FUNCTION_BLOCK F_GetItemAITests EXTENDS TcUnit.FB_TestSuite

VAR
	
	(* In/Out test*)		
	
END_VAR



//==============================================================
//01.CASE_Code
//==============================================================
Case_code01_GTIN_extractedWrong();
Case_code02_SERIAL_extractedWrong();
Case_code03_RSKU_extractedWrong();
Case_code04_BATCH_extractedWrong();
Case_code05_PO_extractedWrong();

//==============================================================
//02.Outer_Code
//==============================================================


//==============================================================
//03.Pack_Code
//==============================================================

METHOD INTERNAL Case_code01_GTIN_extractedWrong
VAR
	sFullCode		: T_MaxString;
	eCodeType		: CODE.E_CodeAI;
	stCodeInfo		: CODE.ST_CodeInfo;
	
	sF_GetItemAI	: T_MaxString;	
END_VAR
// Validation data init
stCodeInfo.eCodeType	:= CODE.E_CodeType.E_CASE;
TestInit(eCodeType := eCodeType, sFullCode := sFullcode, stCodeInfo := stCodeInfo);

//Change some data for test scenario below
sFullCode := '(01)17501031711052(21)86174He081137058500(240)10108245(10)86352024(91)5304012';
eCodeType	:= CODE.E_CodeAI.GTIN;


	
TcUnit.TEST('Case_code01_GTIN_extractedWrong');

	sF_GetItemAI := CODE.F_GetItemAI(sFullCode := sFullCode, 
									 eCodeType := eCodeType, 
									 stCodeInfo := stCodeInfo);
	
	AssertEquals_STRING(Expected:= '17501031711052', 
						Actual:= TO_STRING(sF_GetItemAI), 
						Message:= 'Wrong GTIN extracted');						

TEST_FINISHED();
END_METHOD

METHOD INTERNAL Case_code02_SERIAL_extractedWrong
VAR
	sFullCode		: T_MaxString;
	eCodeType		: CODE.E_CodeAI;
	stCodeInfo		: CODE.ST_CodeInfo;
	
	sF_GetItemAI	: T_MaxString;	
END_VAR
// Validation data init
stCodeInfo.eCodeType	:= CODE.E_CodeType.E_CASE;
TestInit(eCodeType := eCodeType, sFullCode := sFullcode, stCodeInfo := stCodeInfo);

//Change some data for test scenario below
sFullCode := '(01)17501031711052(21)86174He081137058500(240)10108245(10)86352024(91)5304012';
eCodeType	:= CODE.E_CodeAI.SERIAL;


	
TcUnit.TEST('Case_code02_SERIAL_extractedWrong');

	sF_GetItemAI := CODE.F_GetItemAI(sFullCode := sFullCode, 
									 eCodeType := eCodeType, 
									 stCodeInfo := stCodeInfo);
	
	AssertEquals_STRING(Expected:= '86174He081137058500', 
						Actual:= TO_STRING(sF_GetItemAI), 
						Message:= 'Wrong SERIAL extracted');						

TEST_FINISHED();
END_METHOD

METHOD INTERNAL Case_code03_RSKU_extractedWrong
VAR
	sFullCode		: T_MaxString;
	eCodeType		: CODE.E_CodeAI;
	stCodeInfo		: CODE.ST_CodeInfo;
	
	sF_GetItemAI	: T_MaxString;	
END_VAR
// Validation data init
stCodeInfo.eCodeType	:= CODE.E_CodeType.E_CASE;
TestInit(eCodeType := eCodeType, sFullCode := sFullcode, stCodeInfo := stCodeInfo);

//Change some data for test scenario below
sFullCode := '(01)17501031711052(21)86174He081137058500(240)10108245(10)86352024(91)5304012';
eCodeType	:= CODE.E_CodeAI.RSKU;


	
TcUnit.TEST('Case_code03_RSKU_extractedWrong');

	sF_GetItemAI := CODE.F_GetItemAI(sFullCode := sFullCode, 
									 eCodeType := eCodeType, 
									 stCodeInfo := stCodeInfo);
	
	AssertEquals_STRING(Expected:= '10108245', 
						Actual:= TO_STRING(sF_GetItemAI), 
						Message:= 'Wrong RSKU extracted');						

TEST_FINISHED();
END_METHOD

METHOD INTERNAL Case_code04_BATCH_extractedWrong
VAR
	sFullCode		: T_MaxString;
	eCodeType		: CODE.E_CodeAI;
	stCodeInfo		: CODE.ST_CodeInfo;
	
	sF_GetItemAI	: T_MaxString;	
END_VAR
// Validation data init
stCodeInfo.eCodeType	:= CODE.E_CodeType.E_CASE;
TestInit(eCodeType := eCodeType, sFullCode := sFullcode, stCodeInfo := stCodeInfo);

//Change some data for test scenario below
sFullCode := '(01)17501031711052(21)86174He081137058500(240)10108245(10)86352024(91)5304012';
eCodeType	:= CODE.E_CodeAI.BATCH;


	
TcUnit.TEST('Case_code04_BATCH_extractedWrong');

	sF_GetItemAI := CODE.F_GetItemAI(sFullCode := sFullCode, 
									 eCodeType := eCodeType, 
									 stCodeInfo := stCodeInfo);
	
	AssertEquals_STRING(Expected:= '86352024', 
						Actual:= TO_STRING(sF_GetItemAI), 
						Message:= 'Wrong BATCH extracted');						

TEST_FINISHED();
END_METHOD

METHOD INTERNAL Case_code05_PO_extractedWrong
VAR
	sFullCode		: T_MaxString;
	eCodeType		: CODE.E_CodeAI;
	stCodeInfo		: CODE.ST_CodeInfo;
	
	sF_GetItemAI	: T_MaxString;	
END_VAR
// Validation data init
stCodeInfo.eCodeType	:= CODE.E_CodeType.E_CASE;
TestInit(eCodeType := eCodeType, sFullCode := sFullcode, stCodeInfo := stCodeInfo);

//Change some data for test scenario below
sFullCode := '(01)17501031711052(21)86174He081137058500(240)10108245(10)86352024(91)5304012';
eCodeType	:= CODE.E_CodeAI.PO;


	
TcUnit.TEST('Case_code05_PO_extractedWrong');

	sF_GetItemAI := CODE.F_GetItemAI(sFullCode := sFullCode, 
									 eCodeType := eCodeType, 
									 stCodeInfo := stCodeInfo);
	
	AssertEquals_STRING(Expected:= '5304012', 
						Actual:= TO_STRING(sF_GetItemAI), 
						Message:= 'Wrong PO extracted');						

TEST_FINISHED();
END_METHOD

METHOD PRIVATE TestInit
VAR_IN_OUT
	eCodeType		: CODE.E_CodeAI;
	stCodeInfo		: CODE.ST_CodeInfo;
	sFullCode		: T_MaxString;
END_VAR

VAR	
END_VAR

// Case validation recipe
IF stCodeInfo.eCodeType = CODE.E_CodeType.E_CASE THEN

// GTIN 
	stCodeInfo.stGTIN.sStartAI := '(01)';
	stCodeInfo.stGTIN.sEndAI := '(';
	stCodeInfo.stGTIN.nCodeLength := 14;
	stCodeInfo.stGTIN.nCodeStartPos := 0;	
	
// SERIAL	
	stCodeInfo.stSerialCode.sStartAI := '(21)';
	stCodeInfo.stSerialCode.sEndAI := '(';
	stCodeInfo.stSerialCode.nCodeLength := 19;
	stCodeInfo.stSerialCode.nCodeStartPos := 0;	
	
// RSKU
	stCodeInfo.stRSKU.sStartAI := '(240)';
	stCodeInfo.stRSKU.sEndAI := '(';
	stCodeInfo.stRSKU.nCodeLength := 8;
	stCodeInfo.stRSKU.nCodeStartPos := 0;	
	
// BATCH
	stCodeInfo.stBatchID.sStartAI := '(10)';
	stCodeInfo.stBatchID.sEndAI := '(';
	stCodeInfo.stBatchID.nCodeLength := 8;
	stCodeInfo.stBatchID.nCodeStartPos := 0;	
	
// PRODUCTION ORDER
	stCodeInfo.stProductionOrder.sStartAI := '(91)';
	stCodeInfo.stProductionOrder.sEndAI := '(';
	stCodeInfo.stProductionOrder.nCodeLength := 7;
	stCodeInfo.stProductionOrder.nCodeStartPos := 0;	

stCodeInfo.nMinLength 		:= 10; // NOT used
stCodeInfo.nEntireLength	:= 77;
stCodeInfo.nNumberOfAIs		:= 5;
	
ELSIF stCodeInfo.eCodeType = CODE.E_CodeType.E_OUTER THEN
	;

ELSIF stCodeInfo.eCodeType = CODE.E_CodeType.E_PACK THEN
	;

END_IF
END_METHOD

END_FUNCTION_BLOCK

(* stored: Version 1.1.0.1
   POU F_GetItemAITests: Id {18f97de6-ed76-44ae-ba5e-7b2d44347ddb}, SpecialFunc None
   Folder 01.CASE_Code: Id {eca26ad4-16d4-4352-be9e-83f84f9e1ce9}
   Method Case_code01_GTIN_extractedWrong: Id {f0d30fae-952e-4f2f-ac9d-a35fda3e20c7}
   Method Case_code02_SERIAL_extractedWrong: Id {4e805853-f7f7-4d55-b6fc-937e82a34cb1}
   Method Case_code03_RSKU_extractedWrong: Id {565eff76-fd6e-48d5-9237-3a11b21db441}
   Method Case_code04_BATCH_extractedWrong: Id {564485eb-8d27-44ab-86f0-c4cc8f856032}
   Method Case_code05_PO_extractedWrong: Id {ba6b24d7-e296-48d0-9ff5-85c414b06a2f}
   Method TestInit: Id {4eb8a079-32fd-4185-b10b-fa0b793458cd} *)
